FUNCTION_BLOCK Controller (* Basic Function Block Type *)
  (* Standard: 61499-2 *)
  (* Version 0.0, 4/23/2019, vshatrov, nxtControl GmbH, Template *)
  PACKAGE Main;
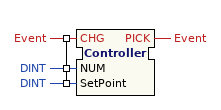
  EVENT_INPUT
    CHG WITH NUM, SetPoint; (* Normal Execution Request *)
  END_EVENT
  EVENT_OUTPUT
    PICK; (* Execution Confirmation *)
  END_EVENT
  VAR_INPUT
    NUM : DINT; (* Input event qualifier *)
    SetPoint : DINT;
  END_VAR
  VAR
    match : BOOL;
  END_VAR
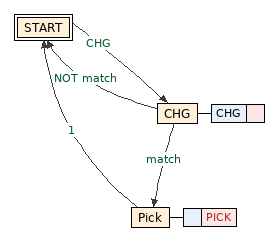
  EC_STATES
    START; (* Initial State *)
    CHG : CHG; (* Normal execution *)
    Pick : -> PICK;
  END_STATES
  EC_TRANSITIONS
    START TO CHG := CHG;
    CHG TO START := NOT match;
    Pick TO START := 1;
    CHG TO Pick := match;
  END_TRANSITIONS
  ALGORITHM CHG IN ST: (* Normally executed algorithm *)
match := NUM = SetPoint;
  END_ALGORITHM
END_FUNCTION_BLOCK
